// TIA Portal project "babu_3wayTrafficLight_Not_India" (V15)

(* hardware
DEVICE "S7-1200 station_1"  S7-1200 Station
   slot 0: "Rack_0"  S7-1200 Rack  Rack  V1.0
   slot 1: "PLC_1"  CPU 1212C DC/DC/DC  6ES7 212-1AE40-0XB0  V4.2
*)

// ===== PLC "PLC_1"  CPU 1212C DC/DC/DC =====

VAR_GLOBAL   // PLC tag table "Default tag table"
   "Push Button" AT %I0.0 : Bool;
   "Push Button Memory" AT %M0.0 : Bool;
   "INITIALIZE" AT %M0.1 : Bool;
   "R1M" AT %M0.2 : Bool;
   "R2M" AT %M0.3 : Bool;
   "R3M" AT %M0.4 : Bool;
   "G1M" AT %M1.0 : Bool;
   "G2M" AT %M1.1 : Bool;
   "G3M" AT %M1.2 : Bool;
   "G3" AT %Q0.0 : Bool;
   "Y1" AT %Q0.1 : Bool;
   "Y1G1M" AT %M1.3 : Bool;
   "Y1R1M" AT %M1.4 : Bool;
   "Y2G2M" AT %M1.5 : Bool;
   "Y2R2M" AT %M1.6 : Bool;
   "Y3R3M" AT %M1.7 : Bool;
   "Y3G3M" AT %M2.0 : Bool;
   "G1" AT %Q0.2 : Bool;
   "Y2" AT %Q0.3 : Bool;
   "G2" AT %Q0.4 : Bool;
END_VAR

// folder: System blocks/Program resources

DATA_BLOCK "IEC_Timer_0_DB"   // DB1
{ S7_Optimized_Access := 'TRUE' }
AUTHOR : Simatic
FAMILY : IEC
NAME : IEC_TMR
VERSION : 1.0
// stored: InstanceOfName IEC_TIMER
"IEC_TIMER"
BEGIN
END_DATA_BLOCK

DATA_BLOCK "IEC_Timer_0_DB_1"   // DB2
{ S7_Optimized_Access := 'TRUE' }
AUTHOR : Simatic
FAMILY : IEC
NAME : IEC_TMR
VERSION : 1.0
// stored: InstanceOfName IEC_TIMER
"IEC_TIMER"
BEGIN
END_DATA_BLOCK

DATA_BLOCK "IEC_Timer_0_DB_2"   // DB3
{ S7_Optimized_Access := 'TRUE' }
AUTHOR : Simatic
FAMILY : IEC
NAME : IEC_TMR
VERSION : 1.0
// stored: InstanceOfName IEC_TIMER
"IEC_TIMER"
BEGIN
END_DATA_BLOCK

DATA_BLOCK "IEC_Timer_0_DB_3"   // DB4
{ S7_Optimized_Access := 'TRUE' }
AUTHOR : Simatic
FAMILY : IEC
NAME : IEC_TMR
VERSION : 1.0
// stored: InstanceOfName IEC_TIMER
"IEC_TIMER"
BEGIN
END_DATA_BLOCK

DATA_BLOCK "IEC_Timer_0_DB_4"   // DB5
{ S7_Optimized_Access := 'TRUE' }
AUTHOR : Simatic
FAMILY : IEC
NAME : IEC_TMR
VERSION : 1.0
// stored: InstanceOfName IEC_TIMER
"IEC_TIMER"
BEGIN
END_DATA_BLOCK

DATA_BLOCK "IEC_Timer_0_DB_5"   // DB6
{ S7_Optimized_Access := 'TRUE' }
AUTHOR : Simatic
FAMILY : IEC
NAME : IEC_TMR
VERSION : 1.0
// stored: InstanceOfName IEC_TIMER
"IEC_TIMER"
BEGIN
END_DATA_BLOCK

DATA_BLOCK "IEC_Timer_0_DB_6"   // DB7
{ S7_Optimized_Access := 'TRUE' }
AUTHOR : Simatic
FAMILY : IEC
NAME : IEC_TMR
VERSION : 1.0
// stored: InstanceOfName IEC_TIMER
"IEC_TIMER"
BEGIN
END_DATA_BLOCK

DATA_BLOCK "IEC_Timer_0_DB_7"   // DB8
{ S7_Optimized_Access := 'TRUE' }
AUTHOR : Simatic
FAMILY : IEC
NAME : IEC_TMR
VERSION : 1.0
// stored: InstanceOfName IEC_TIMER
"IEC_TIMER"
BEGIN
END_DATA_BLOCK

DATA_BLOCK "IEC_Timer_0_DB_8"   // DB9
{ S7_Optimized_Access := 'TRUE' }
AUTHOR : Simatic
FAMILY : IEC
NAME : IEC_TMR
VERSION : 1.0
// stored: InstanceOfName IEC_TIMER
"IEC_TIMER"
BEGIN
END_DATA_BLOCK

DATA_BLOCK "IEC_Timer_0_DB_9"   // DB10
{ S7_Optimized_Access := 'TRUE' }
AUTHOR : Simatic
FAMILY : IEC
NAME : IEC_TMR
VERSION : 1.0
// stored: InstanceOfName IEC_TIMER
"IEC_TIMER"
BEGIN
END_DATA_BLOCK

DATA_BLOCK "IEC_Timer_0_DB_10"   // DB11
{ S7_Optimized_Access := 'TRUE' }
AUTHOR : Simatic
FAMILY : IEC
NAME : IEC_TMR
VERSION : 1.0
// stored: InstanceOfName IEC_TIMER
"IEC_TIMER"
BEGIN
END_DATA_BLOCK

DATA_BLOCK "IEC_Timer_0_DB_11"   // DB12
{ S7_Optimized_Access := 'TRUE' }
AUTHOR : Simatic
FAMILY : IEC
NAME : IEC_TMR
VERSION : 1.0
// stored: InstanceOfName IEC_TIMER
"IEC_TIMER"
BEGIN
END_DATA_BLOCK

DATA_BLOCK "IEC_Timer_0_DB_12"   // DB13
{ S7_Optimized_Access := 'TRUE' }
AUTHOR : Simatic
FAMILY : IEC
NAME : IEC_TMR
VERSION : 1.0
// stored: InstanceOfName IEC_TIMER
"IEC_TIMER"
BEGIN
END_DATA_BLOCK

DATA_BLOCK "IEC_Timer_0_DB_13"   // DB14
{ S7_Optimized_Access := 'TRUE' }
AUTHOR : Simatic
FAMILY : IEC
NAME : IEC_TMR
VERSION : 1.0
// stored: InstanceOfName IEC_TIMER
"IEC_TIMER"
BEGIN
END_DATA_BLOCK

DATA_BLOCK "IEC_Timer_0_DB_14"   // DB15
{ S7_Optimized_Access := 'TRUE' }
AUTHOR : Simatic
FAMILY : IEC
NAME : IEC_TMR
VERSION : 1.0
// stored: InstanceOfName IEC_TIMER
"IEC_TIMER"
BEGIN
END_DATA_BLOCK

DATA_BLOCK "IEC_Timer_0_DB_15"   // DB16
{ S7_Optimized_Access := 'TRUE' }
AUTHOR : Simatic
FAMILY : IEC
NAME : IEC_TMR
VERSION : 1.0
// stored: InstanceOfName IEC_TIMER
"IEC_TIMER"
BEGIN
END_DATA_BLOCK

DATA_BLOCK "IEC_Timer_0_DB_16"   // DB17
{ S7_Optimized_Access := 'TRUE' }
AUTHOR : Simatic
FAMILY : IEC
NAME : IEC_TMR
VERSION : 1.0
// stored: InstanceOfName IEC_TIMER
"IEC_TIMER"
BEGIN
END_DATA_BLOCK

DATA_BLOCK "IEC_Timer_0_DB_17"   // DB18
{ S7_Optimized_Access := 'TRUE' }
AUTHOR : Simatic
FAMILY : IEC
NAME : IEC_TMR
VERSION : 1.0
// stored: InstanceOfName IEC_TIMER
"IEC_TIMER"
BEGIN
END_DATA_BLOCK

DATA_BLOCK "IEC_Timer_0_DB_18"   // DB19
{ S7_Optimized_Access := 'TRUE' }
AUTHOR : Simatic
FAMILY : IEC
NAME : IEC_TMR
VERSION : 1.0
// stored: InstanceOfName IEC_TIMER
"IEC_TIMER"
BEGIN
END_DATA_BLOCK

DATA_BLOCK "IEC_Timer_0_DB_19"   // DB20
{ S7_Optimized_Access := 'TRUE' }
AUTHOR : Simatic
FAMILY : IEC
NAME : IEC_TMR
VERSION : 1.0
// stored: InstanceOfName IEC_TIMER
"IEC_TIMER"
BEGIN
END_DATA_BLOCK

DATA_BLOCK "IEC_Timer_0_DB_20"   // DB21
{ S7_Optimized_Access := 'TRUE' }
AUTHOR : Simatic
FAMILY : IEC
NAME : IEC_TMR
VERSION : 1.0
// stored: InstanceOfName IEC_TIMER
"IEC_TIMER"
BEGIN
END_DATA_BLOCK

DATA_BLOCK "IEC_Timer_0_DB_21"   // DB22
{ S7_Optimized_Access := 'TRUE' }
AUTHOR : Simatic
FAMILY : IEC
NAME : IEC_TMR
VERSION : 1.0
// stored: InstanceOfName IEC_TIMER
"IEC_TIMER"
BEGIN
END_DATA_BLOCK

DATA_BLOCK "IEC_Timer_0_DB_22"   // DB23
{ S7_Optimized_Access := 'TRUE' }
AUTHOR : Simatic
FAMILY : IEC
NAME : IEC_TMR
VERSION : 1.0
// stored: InstanceOfName IEC_TIMER
"IEC_TIMER"
BEGIN
END_DATA_BLOCK

DATA_BLOCK "IEC_Timer_0_DB_23"   // DB24
{ S7_Optimized_Access := 'TRUE' }
AUTHOR : Simatic
FAMILY : IEC
NAME : IEC_TMR
VERSION : 1.0
// stored: InstanceOfName IEC_TIMER
"IEC_TIMER"
BEGIN
END_DATA_BLOCK

DATA_BLOCK "IEC_Timer_0_DB_24"   // DB25
{ S7_Optimized_Access := 'TRUE' }
AUTHOR : Simatic
FAMILY : IEC
NAME : IEC_TMR
VERSION : 1.0
// stored: InstanceOfName IEC_TIMER
"IEC_TIMER"
BEGIN
END_DATA_BLOCK

DATA_BLOCK "IEC_Timer_0_DB_25"   // DB26
{ S7_Optimized_Access := 'TRUE' }
AUTHOR : Simatic
FAMILY : IEC
NAME : IEC_TMR
VERSION : 1.0
// stored: InstanceOfName IEC_TIMER
"IEC_TIMER"
BEGIN
END_DATA_BLOCK

DATA_BLOCK "IEC_Timer_0_DB_26"   // DB27
{ S7_Optimized_Access := 'TRUE' }
AUTHOR : Simatic
FAMILY : IEC
NAME : IEC_TMR
VERSION : 1.0
// stored: InstanceOfName IEC_TIMER
"IEC_TIMER"
BEGIN
END_DATA_BLOCK

DATA_BLOCK "IEC_Timer_0_DB_27"   // DB28
{ S7_Optimized_Access := 'TRUE' }
AUTHOR : Simatic
FAMILY : IEC
NAME : IEC_TMR
VERSION : 1.0
// stored: InstanceOfName IEC_TIMER
"IEC_TIMER"
BEGIN
END_DATA_BLOCK

// folder: (top level)

ORGANIZATION_BLOCK "Main"   // OB1, LAD, ProgramCycle
TITLE = "Main Program Sweep (Cycle)"
{ S7_Optimized_Access := 'TRUE' }
VERSION : 0.1
   VAR_INPUT
      Initial_Call : Bool;   // Initial call of this OB
      Remanence : Bool;   // =True, if remanent data are available
   END_VAR
   VAR_TEMP   // added for the SCL form of the ladder/FBD networks
      _w1 : Bool;
   END_VAR
BEGIN

REGION Network 1
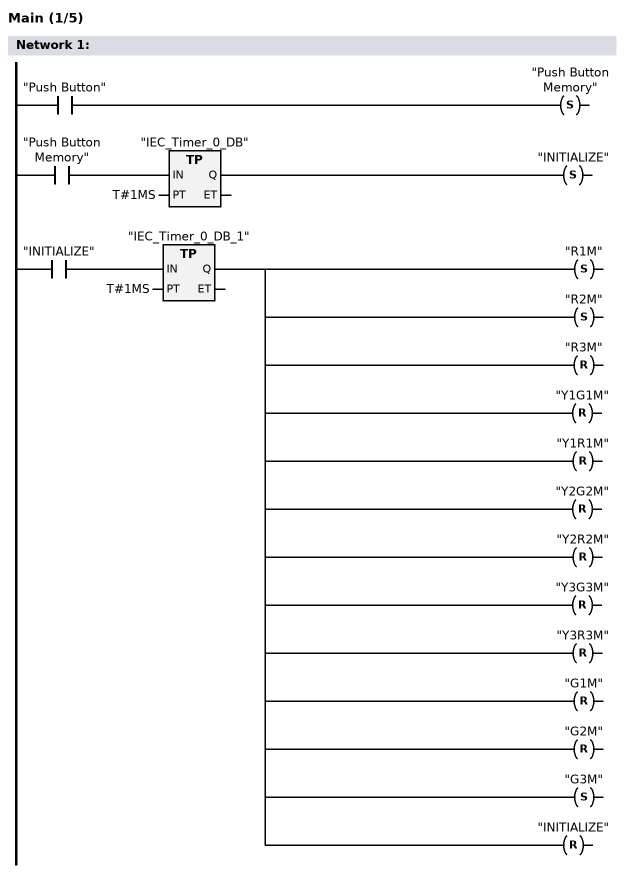
   IF "Push Button" THEN "Push Button Memory" := TRUE; END_IF;
   "IEC_Timer_0_DB".TP(IN := "Push Button Memory", PT := T#1MS);
   IF "IEC_Timer_0_DB".Q THEN "INITIALIZE" := TRUE; END_IF;
   "IEC_Timer_0_DB_1".TP(IN := "INITIALIZE", PT := T#1MS);
   IF "IEC_Timer_0_DB_1".Q THEN
       "R1M" := TRUE;
       "R2M" := TRUE;
       "R3M" := FALSE;
       "Y1G1M" := FALSE;
       "Y1R1M" := FALSE;
       "Y2G2M" := FALSE;
       "Y2R2M" := FALSE;
       "Y3G3M" := FALSE;
       "Y3R3M" := FALSE;
       "G1M" := FALSE;
       "G2M" := FALSE;
       "G3M" := TRUE;
       "INITIALIZE" := FALSE;
   END_IF;
END_REGION

REGION Network 2
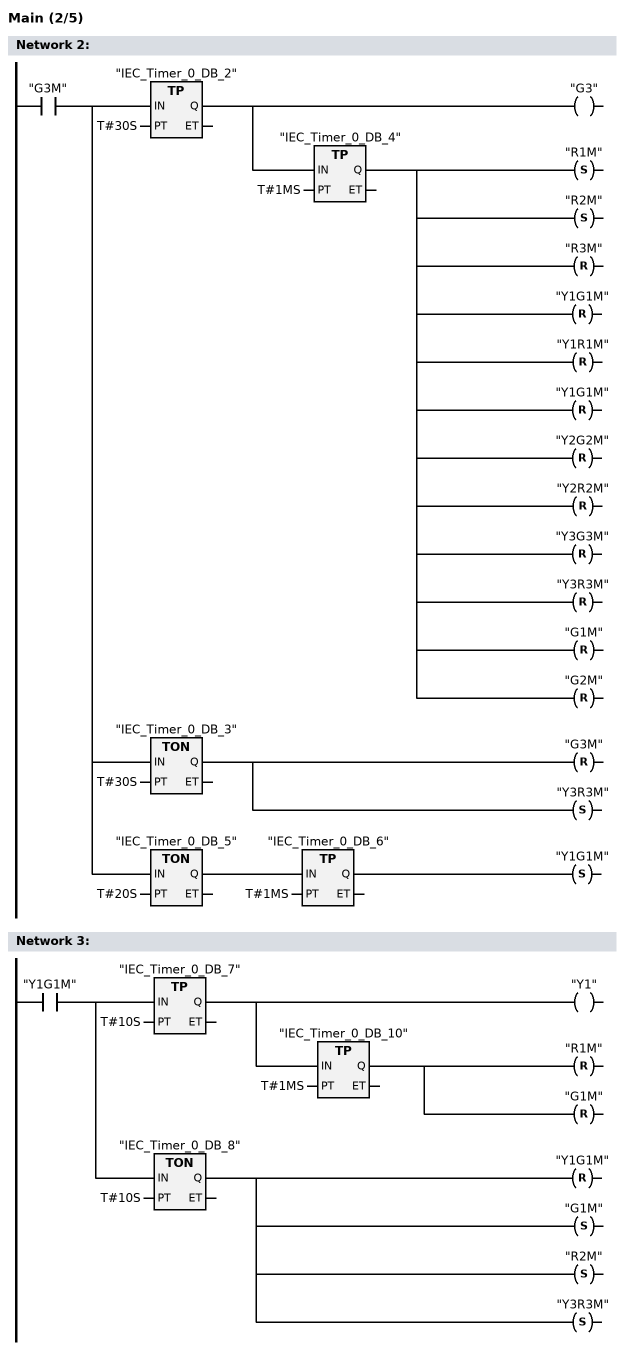
   "IEC_Timer_0_DB_2".TP(IN := "G3M", PT := T#30S);
   "G3" := "IEC_Timer_0_DB_2".Q;
   "IEC_Timer_0_DB_4".TP(IN := "IEC_Timer_0_DB_2".Q, PT := T#1MS);
   IF "IEC_Timer_0_DB_4".Q THEN
       "R1M" := TRUE;
       "R2M" := TRUE;
       "R3M" := FALSE;
       "Y1G1M" := FALSE;
       "Y1R1M" := FALSE;
       "Y1G1M" := FALSE;
       "Y2G2M" := FALSE;
       "Y2R2M" := FALSE;
       "Y3G3M" := FALSE;
       "Y3R3M" := FALSE;
       "G1M" := FALSE;
       "G2M" := FALSE;
   END_IF;
   "IEC_Timer_0_DB_3".TON(IN := "G3M", PT := T#30S);
   #_w1 := "G3M";
   IF "IEC_Timer_0_DB_3".Q THEN
       "G3M" := FALSE;
       "Y3R3M" := TRUE;
   END_IF;
   "IEC_Timer_0_DB_5".TON(IN := #_w1, PT := T#20S);
   "IEC_Timer_0_DB_6".TP(IN := "IEC_Timer_0_DB_5".Q, PT := T#1MS);
   IF "IEC_Timer_0_DB_6".Q THEN "Y1G1M" := TRUE; END_IF;
END_REGION

REGION Network 3
   "IEC_Timer_0_DB_7".TP(IN := "Y1G1M", PT := T#10S);
   "Y1" := "IEC_Timer_0_DB_7".Q;
   "IEC_Timer_0_DB_10".TP(IN := "IEC_Timer_0_DB_7".Q, PT := T#1MS);
   IF "IEC_Timer_0_DB_10".Q THEN
       "R1M" := FALSE;
       "G1M" := FALSE;
   END_IF;
   "IEC_Timer_0_DB_8".TON(IN := "Y1G1M", PT := T#10S);
   IF "IEC_Timer_0_DB_8".Q THEN
       "Y1G1M" := FALSE;
       "G1M" := TRUE;
       "R2M" := TRUE;
       "Y3R3M" := TRUE;
   END_IF;
END_REGION

REGION Network 4
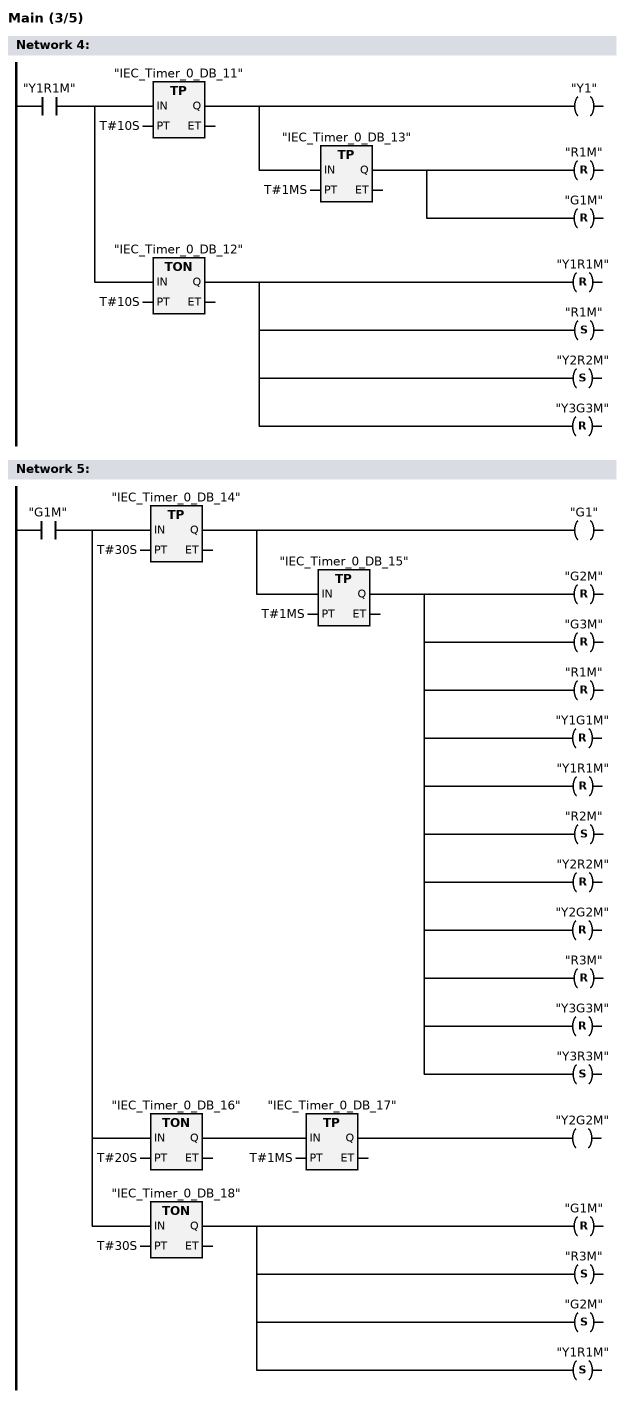
   "IEC_Timer_0_DB_11".TP(IN := "Y1R1M", PT := T#10S);
   "Y1" := "IEC_Timer_0_DB_11".Q;
   "IEC_Timer_0_DB_13".TP(IN := "IEC_Timer_0_DB_11".Q, PT := T#1MS);
   IF "IEC_Timer_0_DB_13".Q THEN
       "R1M" := FALSE;
       "G1M" := FALSE;
   END_IF;
   "IEC_Timer_0_DB_12".TON(IN := "Y1R1M", PT := T#10S);
   IF "IEC_Timer_0_DB_12".Q THEN
       "Y1R1M" := FALSE;
       "R1M" := TRUE;
       "Y2R2M" := TRUE;
       "Y3G3M" := FALSE;
   END_IF;
END_REGION

REGION Network 5
   "IEC_Timer_0_DB_14".TP(IN := "G1M", PT := T#30S);
   "G1" := "IEC_Timer_0_DB_14".Q;
   "IEC_Timer_0_DB_15".TP(IN := "IEC_Timer_0_DB_14".Q, PT := T#1MS);
   IF "IEC_Timer_0_DB_15".Q THEN
       "G2M" := FALSE;
       "G3M" := FALSE;
       "R1M" := FALSE;
       "Y1G1M" := FALSE;
       "Y1R1M" := FALSE;
       "R2M" := TRUE;
       "Y2R2M" := FALSE;
       "Y2G2M" := FALSE;
       "R3M" := FALSE;
       "Y3G3M" := FALSE;
       "Y3R3M" := TRUE;
   END_IF;
   "IEC_Timer_0_DB_16".TON(IN := "G1M", PT := T#20S);
   "IEC_Timer_0_DB_17".TP(IN := "IEC_Timer_0_DB_16".Q, PT := T#1MS);
   "Y2G2M" := "IEC_Timer_0_DB_17".Q;
   "IEC_Timer_0_DB_18".TON(IN := "G1M", PT := T#30S);
   IF "IEC_Timer_0_DB_18".Q THEN
       "G1M" := FALSE;
       "R3M" := TRUE;
       "G2M" := TRUE;
       "Y1R1M" := TRUE;
   END_IF;
END_REGION

REGION Network 6
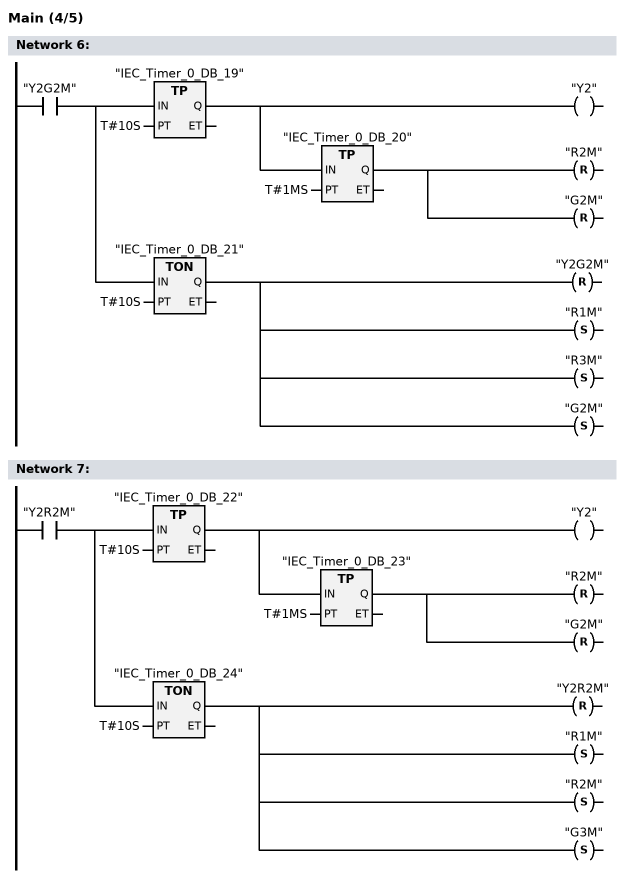
   "IEC_Timer_0_DB_19".TP(IN := "Y2G2M", PT := T#10S);
   "Y2" := "IEC_Timer_0_DB_19".Q;
   "IEC_Timer_0_DB_20".TP(IN := "IEC_Timer_0_DB_19".Q, PT := T#1MS);
   IF "IEC_Timer_0_DB_20".Q THEN
       "R2M" := FALSE;
       "G2M" := FALSE;
   END_IF;
   "IEC_Timer_0_DB_21".TON(IN := "Y2G2M", PT := T#10S);
   IF "IEC_Timer_0_DB_21".Q THEN
       "Y2G2M" := FALSE;
       "R1M" := TRUE;
       "R3M" := TRUE;
       "G2M" := TRUE;
   END_IF;
END_REGION

REGION Network 7
   "IEC_Timer_0_DB_22".TP(IN := "Y2R2M", PT := T#10S);
   "Y2" := "IEC_Timer_0_DB_22".Q;
   "IEC_Timer_0_DB_23".TP(IN := "IEC_Timer_0_DB_22".Q, PT := T#1MS);
   IF "IEC_Timer_0_DB_23".Q THEN
       "R2M" := FALSE;
       "G2M" := FALSE;
   END_IF;
   "IEC_Timer_0_DB_24".TON(IN := "Y2R2M", PT := T#10S);
   IF "IEC_Timer_0_DB_24".Q THEN
       "Y2R2M" := FALSE;
       "R1M" := TRUE;
       "R2M" := TRUE;
       "G3M" := TRUE;
   END_IF;
END_REGION

REGION Network 8
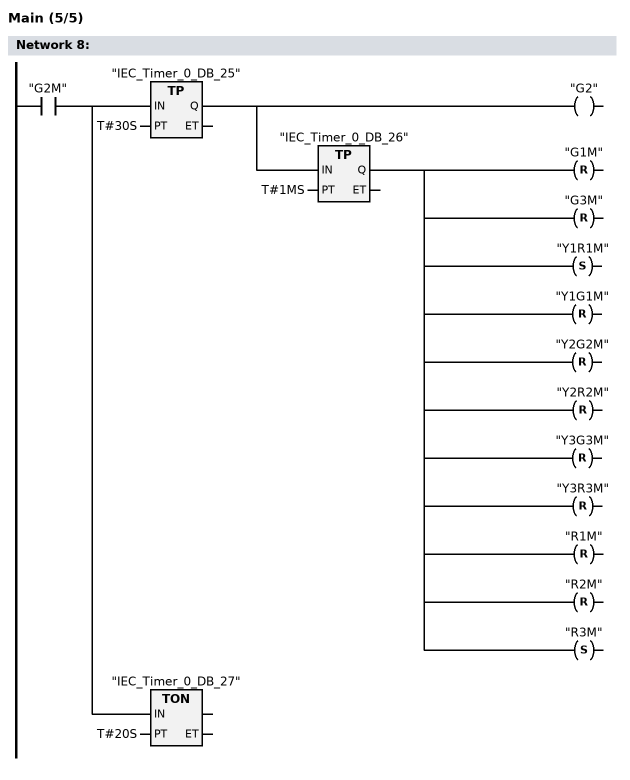
   "IEC_Timer_0_DB_25".TP(IN := "G2M", PT := T#30S);
   "G2" := "IEC_Timer_0_DB_25".Q;
   "IEC_Timer_0_DB_26".TP(IN := "IEC_Timer_0_DB_25".Q, PT := T#1MS);
   IF "IEC_Timer_0_DB_26".Q THEN
       "G1M" := FALSE;
       "G3M" := FALSE;
       "Y1R1M" := TRUE;
       "Y1G1M" := FALSE;
       "Y2G2M" := FALSE;
       "Y2R2M" := FALSE;
       "Y3G3M" := FALSE;
       "Y3R3M" := FALSE;
       "R1M" := FALSE;
       "R2M" := FALSE;
       "R3M" := TRUE;
   END_IF;
   "IEC_Timer_0_DB_27".TON(IN := "G2M", PT := T#20S);
END_REGION
END_ORGANIZATION_BLOCK